// Mitsubishi GX Works2 project: LRI - Lógica Contato de selo   PLC: Q03UDV
// HelloWorld

PROGRAM MAIN
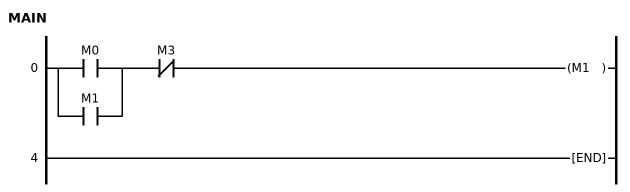
0     LD      M0
      OR      M1
      ANI     M3
      OUT     M1
4     END
END_PROGRAM
